// TIA Portal V20 export
FUNCTION_BLOCK "FB_StatusPart"   // FB87, SCL
{ S7_Optimized_Access := 'TRUE' }
// stored: MemoryReserve 100, SetENOAutomatically false
   VAR_INPUT
      iGood { ExternalAccessible := 'False'; ExternalVisible := 'False'; ExternalWritable := 'False'} : Bool;
      iUnknown { ExternalAccessible := 'False'; ExternalVisible := 'False'; ExternalWritable := 'False'} : Bool;
      iBad { ExternalAccessible := 'False'; ExternalVisible := 'False'; ExternalWritable := 'False'} : Bool;
      iAbsent { ExternalAccessible := 'False'; ExternalVisible := 'False'; ExternalWritable := 'False'} : Bool;
      iPresentUnexpected { ExternalAccessible := 'False'; ExternalVisible := 'False'; ExternalWritable := 'False'} : Bool;
      iAbsentUnexpected { ExternalAccessible := 'False'; ExternalVisible := 'False'; ExternalWritable := 'False'} : Bool;
   END_VAR
   VAR_OUTPUT
      oStatus { ExternalAccessible := 'False'; ExternalVisible := 'False'; ExternalWritable := 'False'} : "UDT_PartState";
   END_VAR
   VAR CONSTANT
      GOOD : Byte := 3;
      UNKNOW : Byte := 1;
      BAD : Byte := 2;
      ABSENT : Byte := 0;
      PRESENT_UNEXPECTED : Byte := 4;
      ABSENT_UNEXPECTED : Byte := 5;
      UNKNOW_STATUS : Byte := 99;
   END_VAR
BEGIN
   REGION Description header 
       //==================================================================================
       // POSALUX Swiss SA / (C) Copyright 2024
       //----------------------------------------------------------------------------------
       // Title: FB_StatusPart
       // Comment/Function: 
       //
       // Author: Fabien WALDT
       // Engineering: TIA Portal v20
       //----------------------------------------------------------------------------------
       // Change log table:
       // Version  | Date     | Expert in charge | Changes applied
       // ---------|----------|------------------|------------------------------------
       // 00.00.01 | 20251024 | WFA              | First released version
       // ==================================================================================
   END_REGION

   REGION Status
       #oStatus.Good := #iGood;
       #oStatus.Unknown := #iUnknown;
       #oStatus.Bad := #iBad;
       #oStatus.Absent := #iAbsent;
       #oStatus.PresentUnexpected := #iPresentUnexpected;
       #oStatus.AbsentUnexpected := #iAbsentUnexpected;
   END_REGION
END_FUNCTION_BLOCK
